(* CoDeSys 2.3 export: TO_SEC.EXP *)

(* POU FUNv1/TO_SEC, ST *)
FUNCTION TO_SEC : TIME
VAR_INPUT
	in: DWORD;
END_VAR
VAR
END_VAR
TO_SEC := DWORD_TO_TIME(in)*1000;
END_FUNCTION
